Staubli VAL3: place_f2.pgx

program place_f2()
begin
  //safe height
  //place
  //shut off
  dDio_t1_vg = off
  //back with blow

end
